// TIA Portal V20 export
TYPE "HMIAxisCtrl_typeActualValues"
TITLE = HMIAxisCtrl_typeActualValues
// Support: tech.team.motioncontrol@siemens.com 
// Fax: +49 (0) 9131/98-1297
   STRUCT
      actualVelocity : LReal;   // Actual value of velocity
      actualPosition : LReal;   // Actual value of position
      targetPosition : LReal;   // Actual value of target position
      isHomed : Bool;   // TRUE: Axis is homed
      brakeIsOpen : Bool;   // TRUE: Brake is open
      axisAlarm : UDInt;   // Number of the technology alarm
      axisError : Bool;   // TRUE: Axis has error
      errorDetailReaction : DInt;   // Effective alarm reaction
   END_STRUCT;
END_TYPE
